# B&R Automation Studio project lab2
Automation Studio 4.5.2.102

## Configuration SampleText

### Task classes (Cpu.sw)
```
Cyclic#4 (cycle 2000 us, tolerance 2000 us):
  Program <- Program.prg
Binaries: TCData, ashwd, User, asfw, arconfig, sysconf, Role, iomap
Libraries: sys_lib, Runtime, asstring, DriveLib
```

### Hardware
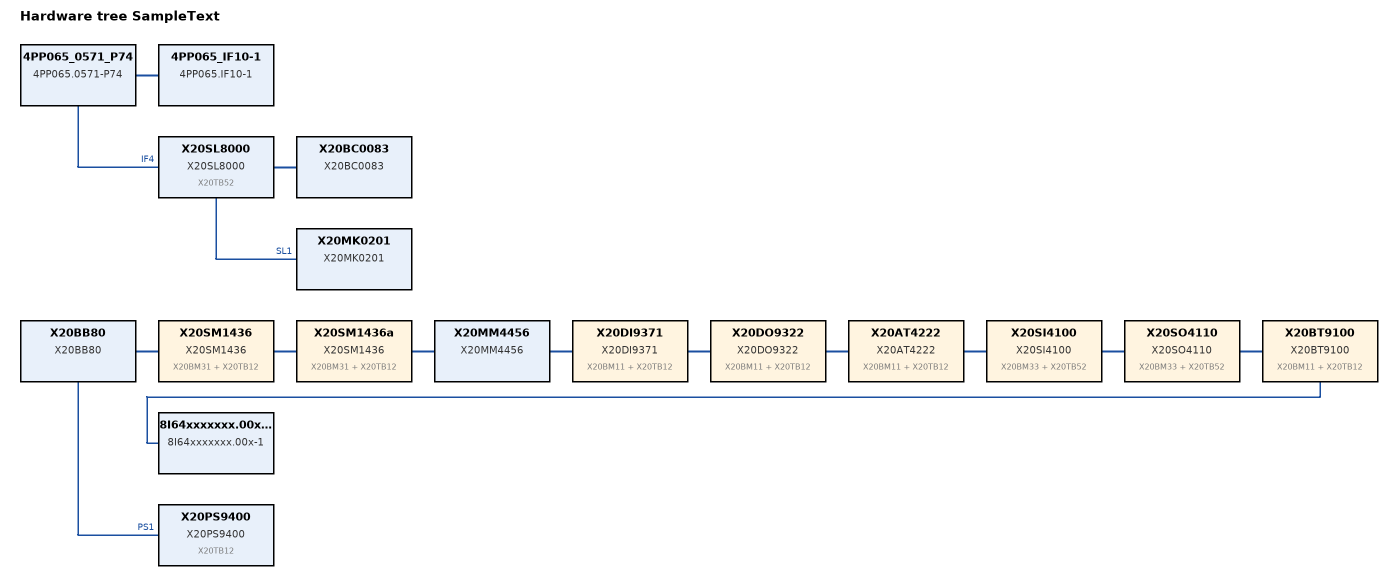
```
4PP065_0571_P74 : 4PP065.0571-P74 v1.1.2.0
  Connector IF4:
    EplInterfaceRedundant = 0
    EplEthInterfaceRedundant = 0
  Connector IF5:
    ActivateDevice = 1
    Mode = Manual
    InternetAddress = 10.0.1.10
    SubnetMask = 255.255.255.0
  ConfigurationID = labBR
  TimerDeviceType = EPLX2X
  TimerDevice = 4PP065_0571_P74.IF4
  TaskClassIdleTime = 2000
  Cyclic1Duration = 100000
  Cyclic1Tolerance = 0
  Cyclic1Output = 1
  Cyclic4Duration = 2000
  Cyclic4Tolerance = 2000
4PP065_IF10-1 : 4PP065.IF10-1 v1.0.3.0  [SS -> 4PP065_0571_P74.SS1]
8I64xxxxxxx.00x-1 : 8I64xxxxxxx.00x-1 v1.3.9.1  [X2X1 -> X20BT9100.X2X1 [Cable Type=X2XCable, Length=10, Version=1.0.0.2]]
  FunctionModel = Standard
  packedETAD = packed
  packedETI = packed
  packedCMDD = packed
  packedCMI = packed
  UNS = 220
  NCR = 10
  NSP = 890
  COS = 64
  RSC = 33000
X20AT4222 : X20AT4222 v1.2.3.0  [SS1 -> X20TB12e.SS; SL -> X20BM11c.SL1]
X20BB80 : X20BB80 v1.0.2.0
X20BC0083 : X20BC0083 v2.7.0.0  [PLK1 -> X20SL8000.PLK2 (NodeNumber=2) [Cable Type=PowerlinkCable, Length=10, Version=1.0.0.2]; SL -> X20BB80.SL1]
X20BM11 : X20BM11 v1.0.0.1  [X2X1 -> X20BM33a.X2X2]
X20BM11a : X20BM11 v1.0.0.1  [X2X1 -> X20MM4456.X2X2]
X20BM11b : X20BM11 v1.0.0.1  [X2X1 -> X20BM11a.X2X2]
X20BM11c : X20BM11 v1.0.0.1  [X2X1 -> X20BM11b.X2X2]
X20BM31 : X20BM31 v1.0.0.1  [X2X1 -> X20BB80.IF1]
X20BM31a : X20BM31 v1.0.0.1  [X2X1 -> X20BM31.X2X2]
X20BM33 : X20BM33 v1.0.0.4  [X2X1 -> X20BM11c.X2X2]
X20BM33a : X20BM33 v1.0.0.4  [X2X1 -> X20BM33.X2X2]
X20BT9100 : X20BT9100 v1.0.3.0  [SS1 -> X20TB12f.SS; SL -> X20BM11.SL1]
X20DI9371 : X20DI9371 v1.0.2.0  [SS1 -> X20TB12c.SS; SL -> X20BM11a.SL1]
X20DO9322 : X20DO9322 v1.0.3.0  [SS1 -> X20TB12d.SS; SL -> X20BM11b.SL1]
X20MK0201 : X20MK0201 v1.0.0.0  [SL -> X20SL8000.SL1]
X20MM4456 : X20MM4456 v1.1.5.0  [X2X1 -> X20BM31a.X2X2]
X20PS9400 : X20PS9400 v1.0.2.4  [SS1 -> X20TB12.SS; PS -> X20BB80.PS1]
X20SI4100 : X20SI4100 v1.10.1.1  [SS1 -> X20TB52.SS; SL -> X20BM33.SL1]
X20SL8000 : X20SL8000 v1.6.5.1  [PLK1 -> 4PP065_0571_P74.IF4 (NodeNumber=1) [Cable Type=PowerlinkCable, Length=10, Version=1.0.0.2]; PLK2 -> X20BC0083.PLK1 (NodeNumber=1) [Cable Type=PowerlinkCable, Length=10, Version=1.0.0.2]; SS1 -> X20TB52b.SS]
  SafeProject = SafeLOGIC-1
X20SM1436 : X20SM1436 v1.4.2.1  [SS1 -> X20TB12a.SS; SL -> X20BM31.SL1]
X20SM1436a : X20SM1436 v1.4.2.1  [SS1 -> X20TB12b.SS; SL -> X20BM31a.SL1]
X20SO4110 : X20SO4110 v1.10.1.1  [SS1 -> X20TB52a.SS; SL -> X20BM33a.SL1]
  SafeModuleID = 3
X20TB12 : X20TB12 v1.0.0.0
X20TB12a : X20TB12 v1.0.0.0
X20TB12b : X20TB12 v1.0.0.0
X20TB12c : X20TB12 v1.0.0.0
X20TB12d : X20TB12 v1.0.0.0
X20TB12e : X20TB12 v1.0.0.0
X20TB12f : X20TB12 v1.0.0.0
X20TB52 : X20TB52 v1.0.0.1
X20TB52a : X20TB52 v1.0.0.1
X20TB52b : X20TB52 v1.0.0.1
```

### IoMap.iom - 4PP065_0571_P74/IoMap.iom
```iecst
VAR_CONFIG
	::Program:doorSM.sw3 AT %IX."X20DI9371".DigitalInput02;
	::Program:doorSM.sw2 AT %IX."X20DI9371".DigitalInput03;
	::Program:doorSM.sw1 AT %IX."X20DI9371".DigitalInput04;
	::Program:doorSM.sw0 AT %IX."X20DI9371".DigitalInput05;
	::Program:ledSM.led3 AT %QX."X20DO9322".DigitalOutput02;
	::Program:ledSM.led2 AT %QX."X20DO9322".DigitalOutput03;
	::Program:ledSM.led1 AT %QX."X20DO9322".DigitalOutput04;
	::Program:ledSM.led0 AT %QX."X20DO9322".DigitalOutput05;
	::Program:doorSM.direction AT %IX."X20DI9371".DigitalInput01;
	::Program:driveSM.state AT %IW."8I64xxxxxxx.00x-1".ETAD_Input;
	::Program:driveSM.command AT %QW."8I64xxxxxxx.00x-1".CMDD_Output;
	::Program:driveSM.speed AT %QW."8I64xxxxxxx.00x-1".LFRD_Output;
	::Program:speed_feedback AT %IW."8I64xxxxxxx.00x-1".RFRD_Input;
END_VAR
```

## Logical view

### Library Logical/DriveLib (ANSIC)

#### Types.typ
```iecst
TYPE
	DoorStates :
		(
		ST_INIT, (*Инициализация параметров и ожидание включения частотного преобразователя*)
		ST_UNKNOWN, (*Ворота в неизвестном положении*)
		ST_OPEN, (*Ворота открыты*)
		ST_CLOSE, (*Ворота закрыты*)
		ST_ACC_POS, (*Ускорение ворот в сторону открытия*)
		ST_ACC_NEG, (*Ускорение ворот в сторону закрытия*)
		ST_POS, (*Движение к открытию*)
		ST_NEG, (*Движение к закрытию*)
		ST_DEC_POS, (*Замедление ворот в сторону открытия*)
		ST_DEC_NEG (*Замедление ворот в сторону закрытия*)
		);
END_TYPE
```

#### Constants.var
```iecst
VAR CONSTANT
	STATE_DISABLED : USINT := 64; (*Система выключена*)
	STATE_READY : USINT := 33; (*Система готова к работе*)
	STATE_SWITCHED_ON : USINT := 35; (*Система работает*)
	CMD_SHUTDOWN : USINT := 6; (*Выключить двигатель*)
	CMD_ENABLED : USINT := 15; (*Приготовиться к работе*)
	CMD_SWITCHED_ON : USINT := 7; (*Выключить двигатель*)
END_VAR
```

#### DriveLib.fun
```iecst
{REDUND_ERROR} {REDUND_UNREPLICABLE} FUNCTION_BLOCK DriveStateMachine (*TODO: Add your comment here*) (*$GROUP=User,$CAT=User,$GROUPICON=User.png,$CATICON=User.png*)
	VAR_INPUT
		state : {REDUND_UNREPLICABLE} UINT; (*Состояние частотног преобразователя*)
		enable : {REDUND_UNREPLICABLE} BOOL; (*Сигнал работы функционального блока*)
	END_VAR
	VAR_OUTPUT
		command : {REDUND_UNREPLICABLE} UINT; (*Команда, подаваемая на частотный преобразователь*)
		speed : {REDUND_UNREPLICABLE} INT; (*Заданная скорость*)
	END_VAR
END_FUNCTION_BLOCK

{REDUND_ERROR} {REDUND_UNREPLICABLE} FUNCTION_BLOCK DoorStateMachine (*TODO: Add your comment here*) (*$GROUP=User,$CAT=User,$GROUPICON=User.png,$CATICON=User.png*)
	VAR_INPUT
		state : {REDUND_UNREPLICABLE} DoorStates; (*Состояние частотного преобразователя*)
		sw0 : {REDUND_UNREPLICABLE} BOOL; (*Сигнал концевого выключателя 1*)
		sw1 : {REDUND_UNREPLICABLE} BOOL; (*Сигнал концевого выключателя 2*)
		sw2 : {REDUND_UNREPLICABLE} BOOL; (*Сигнал концевого выключателя 3*)
		sw3 : {REDUND_UNREPLICABLE} BOOL; (*Сигнал концевого выключателя 4*)
		direction : {REDUND_UNREPLICABLE} BOOL; (*Команда, подаваемая на частотный преобразователь*)
	END_VAR
	VAR_OUTPUT
		speed : {REDUND_UNREPLICABLE} INT; (*Заданная скорость*)
	END_VAR
	VAR
		sw0_prev : {REDUND_UNREPLICABLE} BOOL;
		sw1_prev : {REDUND_UNREPLICABLE} BOOL;
		sw2_prev : {REDUND_UNREPLICABLE} BOOL;
		sw3_prev : {REDUND_UNREPLICABLE} BOOL;
	END_VAR
END_FUNCTION_BLOCK

{REDUND_ERROR} {REDUND_UNREPLICABLE} FUNCTION_BLOCK LedStateMachine (*TODO: Add your comment here*) (*$GROUP=User,$CAT=User,$GROUPICON=User.png,$CATICON=User.png*)
	VAR_INPUT
		state : {REDUND_UNREPLICABLE} UINT; (*Состояние частотного преобразователя*)
	END_VAR
	VAR_OUTPUT
		led0 : {REDUND_UNREPLICABLE} BOOL; (*Сигнал работы функционального блока*)
		led1 : {REDUND_UNREPLICABLE} BOOL; (*Сигнал работы функционального блока*)
		led2 : {REDUND_UNREPLICABLE} BOOL; (*Сигнал работы функционального блока*)
		led3 : {REDUND_UNREPLICABLE} BOOL; (*Сигнал работы функционального блока*)
		timer : {REDUND_UNREPLICABLE} INT; (*Заданная скорость*)
	END_VAR
END_FUNCTION_BLOCK
```

#### DoorStateMachine.c
```c
#include <bur/plctypes.h>
#ifdef __cplusplus
	extern "C"
	{
#endif
	#include "DriveLib.h"
#ifdef __cplusplus
	};
#endif
/* TODO: Add your comment here */
void DoorStateMachine(struct DoorStateMachine* inst)
{
	switch (inst->state){
		case ST_INIT:
			{
				if (inst->direction == 0)
					inst->speed = -100; //max = 890
				else
					inst->speed = 100;
				inst->state = ST_UNKNOWN;
				break;
			}

		case ST_UNKNOWN:
			{
				if (inst->direction == 1 && inst->sw0 != inst->sw0_prev){
					inst->speed = 0;
					inst->state = ST_OPEN;
					inst->sw0_prev = inst->sw0;
				}
				if (inst->direction == 0 && inst->sw3 != inst->sw3_prev){
					inst->speed = 0;
					inst->state = ST_CLOSE;
					inst->sw3_prev = inst->sw3;
				}
				break;
			}

		case ST_OPEN:
			{
				if (inst->direction == 0){
					inst->speed = 100;
					inst->state = ST_ACC_POS;
				}
				break;
			}

		case ST_ACC_POS:
			{
				if (inst->sw1 != inst->sw1_prev){
					inst->speed = 500;
					inst->state = ST_POS;
					inst->sw1_prev = inst->sw1;
				}

				if (inst->direction == 1){
					inst->speed = -100;
					inst->state = ST_DEC_NEG;
				}
				break;
			}

		case ST_POS:
			{
				if (inst->sw2 != inst->sw2_prev){
					inst->speed = 100;
					inst->state = ST_DEC_POS;
					inst->sw2_prev = inst->sw2;
				}
				if (inst->direction == 1){
					inst->speed = -500;
					inst->state = ST_NEG;
				}
				break;
			}

		case ST_DEC_POS:
			{
				if (inst->sw3 != inst->sw3_prev){
					inst->speed = 0;
					inst->state = ST_CLOSE;
					inst->sw3_prev = inst->sw3;
				}
				if (inst->direction == 1){
					inst->speed = -100;
					inst->state = ST_ACC_NEG;
				}
				break;
			}

		case ST_CLOSE:
			{
				if (inst->direction == 1){
					inst->speed = -100;
					inst->state = ST_ACC_NEG;
				}
				break;
			}

		case ST_ACC_NEG:
			{
				if (inst->sw2 != inst->sw2_prev){
					inst->speed = -500;
					inst->state = ST_NEG;
					inst->sw2_prev = inst->sw2;
				}
				if (inst->direction == 0){
					inst->speed = 100;
					inst->state = ST_DEC_POS;
				}
				break;
			}

		case ST_NEG:
			{
				if (inst->sw1 != inst->sw1_prev){
					inst->speed = -100;
					inst->state = ST_DEC_NEG;
					inst->sw1_prev = inst->sw1;
				}
				if (inst->direction == 0){
					inst->speed = 500;
					inst->state = ST_POS;
				}
				break;
			}

		case ST_DEC_NEG:
			{
				if (inst->sw0 != inst->sw0_prev){
					inst->speed = 0;
					inst->state = ST_OPEN;
					inst->sw0_prev = inst->sw0;
				}
				if (inst->direction == 0){
					inst->speed = 100;
					inst->state = ST_ACC_POS;
				}
				break;
			}
	}
}
```

#### DriveStateMachine.c
```c
#include <bur/plctypes.h>
#ifdef __cplusplus
	extern "C"
	{
#endif
	#include "DriveLib.h"
#ifdef __cplusplus
	};
#endif
/* TODO: Add your comment here */
void DriveStateMachine(struct DriveStateMachine* inst)
{
	UINT mask = inst->state & 0x6f;
	if (!inst->enable)
		inst->command = CMD_SHUTDOWN;
	else
	{
		switch(mask){
			case STATE_DISABLED:
				inst->command = CMD_SHUTDOWN;
				break;

			case STATE_READY:
				inst->command = CMD_ENABLED;
				break;

			case STATE_SWITCHED_ON:
				inst->command = CMD_SWITCHED_ON;
				break;
		}
	}
}
```

#### LedStateMachine.c
```c
#include <bur/plctypes.h>
#ifdef __cplusplus
	extern "C"
	{
#endif
	#include "DriveLib.h"
#ifdef __cplusplus
	};
#endif
/* TODO: Add your comment here */
void LedStateMachine(struct LedStateMachine* inst)
{
	inst->timer++;
	switch(inst->state){
		case ST_INIT:
			{
				inst->led0 = 0;
				inst->led1 = 0;
				inst->led2 = 0;
				inst->led3 = 0;
				break;
			}

		case ST_UNKNOWN:
			{
				if (inst->timer % 250 == 0){
					inst->led0 = !inst->led0;
					inst->led1 = !inst->led1;
					inst->led2 = !inst->led2;
					inst->led3 = !inst->led3;
				}
				break;
			}

		case ST_OPEN:
			{
				inst->led0 = 0;
				inst->led1 = 0;
				inst->led2 = 0;
				inst->led3 = 0;
				break;
			}

		case ST_ACC_POS:
			{
				inst->led0 = 1;
				if (inst->timer % 200 == 0)
					inst->led1 = !inst->led1;
				break;
			}

		case ST_POS:
			{
				inst->led0 = 1;
				inst->led1 = 1;
				if (inst->timer % 40 == 0)
					inst->led2 = !inst->led2;
				break;
			}

		case ST_DEC_POS:
			{
				inst->led0 = 1;
				inst->led1 = 1;
				inst->led2 = 1;
				if (inst->timer % 200 == 0)
					inst->led3 = !inst->led3;
				break;
			}

		case ST_CLOSE:
			{
				inst->led0 = 1;
				inst->led1 = 1;
				inst->led2 = 1;
				inst->led3 = 1;
				break;
			}

		case ST_ACC_NEG:
			{
				inst->led0 = 1;
				inst->led1 = 1;
				if (inst->timer % 200 == 0)
					inst->led2 = !inst->led2;
				inst->led3 = 0;
				break;
			}

		case ST_NEG:
			{
				inst->led0 = 1;
				if (inst->timer % 40 == 0)
					inst->led1 = !inst->led1;
				inst->led2 = 0;
				inst->led3 = 0;
				break;
			}

		case ST_DEC_NEG:
			{
				if (inst->timer % 200 == 0)
					inst->led0 = !inst->led0;
				inst->led1 = 0;
				inst->led2 = 0;
				inst->led3 = 0;
				break;
			}
	}
}
```

### Program Logical/Program (ANSIC)

#### Variables.var
```iecst
VAR
	driveSM : DriveStateMachine := (0);
	doorSM : DoorStateMachine := (0);
	ledSM : LedStateMachine := (0);
	speed_feedback : INT := 0;
END_VAR
```

#### Main.c
```c
#include <bur/plctypes.h>

#ifdef _DEFAULT_INCLUDES
	#include <AsDefault.h>
#endif

void _INIT ProgramInit(void)
{
	doorSM.state = ST_INIT;
	doorSM.sw0_prev = doorSM.sw0;
	doorSM.sw1_prev = doorSM.sw1;
	doorSM.sw2_prev = doorSM.sw2;
	doorSM.sw3_prev = doorSM.sw3;
}

void _CYCLIC ProgramCyclic(void)
{
	DoorStateMachine(&doorSM);
	driveSM.enable = 1;
	driveSM.speed = doorSM.speed;
	LedStateMachine(&ledSM);
	ledSM.state = doorSM.state;
	DriveStateMachine(&driveSM);
}

void _EXIT ProgramExit(void)
{

}
```

Listed in the project but not available here: Logical/Global.typ, Logical/Global.var, Logical/Libraries
